# EPICS substitutions: src/iocdoc/testfiles/iocBoot/ioc495idc/templates/softMotor.substitutions
file "$(STD)/stdApp/Db/softMotor.db"
{
pattern
{P,       SM}
# NPI
{495idc:,  sm1}
{495idc:,  sm2}
{495idc:,  sm3}
{495idc:,  sm4}
{495idc:,  sm5}
{495idc:,  sm6}
{495idc:,  sm7}
{495idc:,  sm8}
{495idc:,  sm9}
{495idc:,  sm10}
# DET
{495idc:,  sm11}
{495idc:,  sm12}
{495idc:,  sm13}
{495idc:,  sm14}
{495idc:,  sm15}
{495idc:,  sm16}
{495idc:,  sm17}
{495idc:,  sm18}
{495idc:,  sm19}
{495idc:,  sm20}
# NES
{495idc:,  sm21}
{495idc:,  sm22}
{495idc:,  sm23}
{495idc:,  sm24}
{495idc:,  sm25}
{495idc:,  sm26}
{495idc:,  sm27}
{495idc:,  sm28}
{495idc:,  sm29}
{495idc:,  sm30}
{495idc:,  sm31}
{495idc:,  sm32}
{495idc:,  sm33}
{495idc:,  sm34}
{495idc:,  sm35}
{495idc:,  sm36}
{495idc:,  sm37}
{495idc:,  sm38}
{495idc:,  sm39}
{495idc:,  sm40}
{495idc:,  sm41}
{495idc:,  sm42}
{495idc:,  sm43}
{495idc:,  sm44}
{495idc:,  sm45}
{495idc:,  sm46}
{495idc:,  sm47}
{495idc:,  sm48}
{495idc:,  sm49}
{495idc:,  sm50}
}
